RoboDK station: Stringer B-Bot1-BOX1.rdk

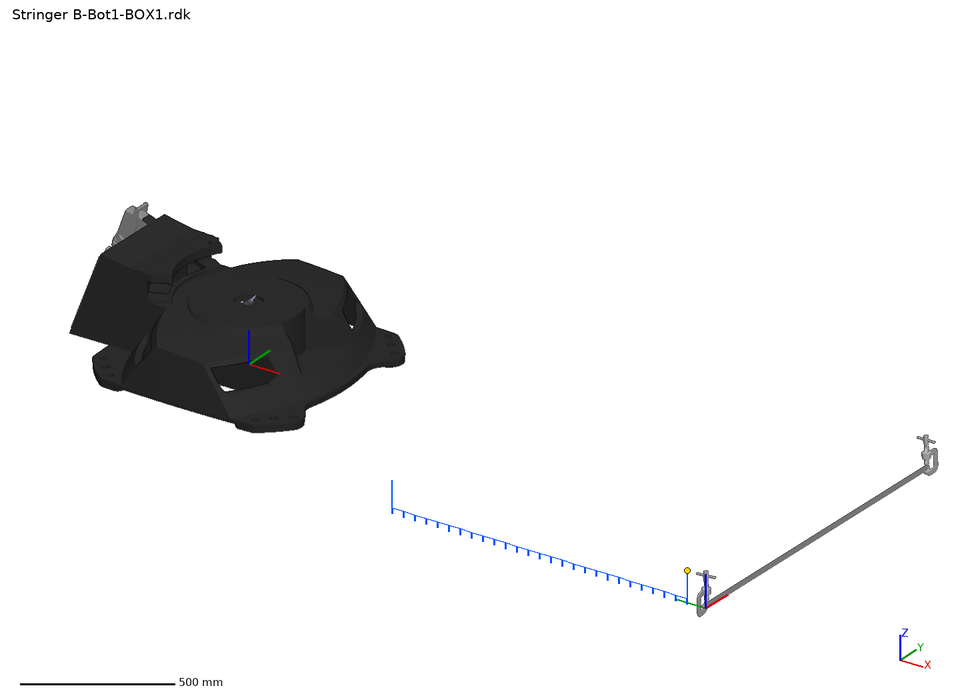
[picture v0: the station drawn from its stored meshes, robots at their saved joint values, targets as dots, program paths as lines]
Station Stringer B-Bot1-BOX1 (saved by RoboDK 5.2.3). Poses are relative to the parent item; angles as X-Y-Z fixed-axis rotations.
  - frame KUKA KR 210 R2700 extra Base at (0, 0, 0) mm
    - robot KUKA KR 210 R2700 extra: 6 axes, payload 210 kg, reach 2696 mm, repeatability 0.06 mm, weight 1068 kg
        joint limits [-185, -140, -120, -350, -125, -350] to [185, -5, 155, 350, 125, 350]; home [0, -90, 90, 0, 0, 0]; saved at [-38.984, -26.717, 86.283, 94.063, 23.385, -126.593]
      - tool Spindle, TCP at (32, 0, 260) mm, rotated rx 0 ry 39 rz 0 deg, size 157.3 x 72 x 259.9 mm
  - frame Frame 2 at (1800, 0, -372.68) mm, rotated rx 0 ry 0 rz 90 deg
    - object STringer B-Bot1-BOX1 at (0, 0, 0) mm, rotated rx 0 ry 0 rz -90 deg, 27 curves, geometry from Point 27
    - object L-Stringer B - Bot1-BOX1 at (0, 0, 0) mm, size 1250 x 20 x 20 mm, geometry from L-Stringer B - Bot1-BOX1.stl
  - machining project Point settings: rotZ(0) | rotX(0)*rotY(0) | rotz(0) | onStart | onPathStart | onApproach | onPoint | onRetract | onFinish | SetRPM(%1) | SetTool(%1) | Extruder(%1) | default | default | OutOnMov(%1) | OutOffMov(%1) | onPathFinish | M_RunCode(%1)
  - program Point (146 instructions, listed below)
  - object FinalClamp at (1791.3, 1250.9, -313.4) mm, rotated rx 0 ry 88.39 rz 0 deg, size 145.3 x 71.1 x 72 mm, geometry from FinalClamp.stp
  - object FinalClamp2 at (1785.63, 21.46, -310.92) mm, rotated rx 159.55 ry 88.7 rz -13.81 deg, size 145.3 x 71.1 x 72 mm, geometry from FinalClamp.stp
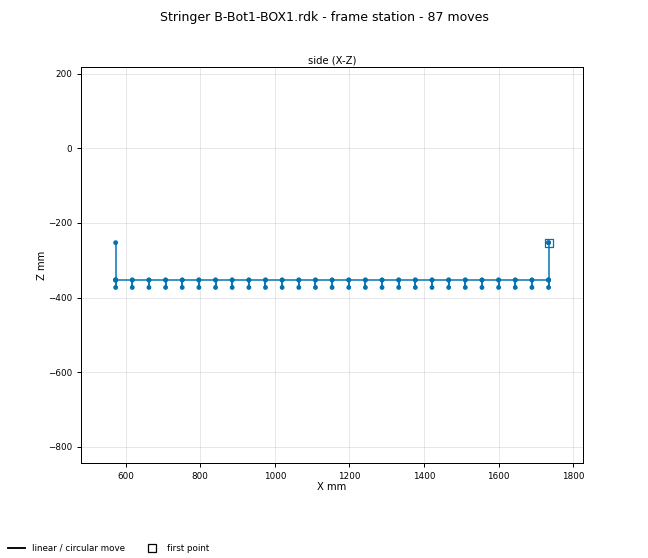
[picture p0: tool path of Stringer B-Bot1-BOX1.rdk in frame station, 87 of 87 moves have a stored position in this frame; points joined in program order, loops and branches not executed]

--- program Point (robot KUKA KR 210 R2700 extra) ---
  Smooth(1)
  Set speed (1000.0 mm/s)
  Set Ref.: Frame 2
  Set Tool: Spindle
  Show Spindle
  MoveJ 1 to (-10.37, 66.57, 120) mm, rotated rx 180 ry 0 rz 180 deg; joints [-2.515, -34.004, 111.796, 176.49, 26.808, -178.821]
  MoveL 2 to (-10.37, 66.57, 120) mm, rotated rx 180 ry 0 rz 180 deg; joints [-2.515, -34.004, 111.796, 176.49, 26.808, -178.821]
  MoveL 3 to (-10.37, 66.57, 20) mm, rotated rx -180 ry 0 rz -180 deg; joints [-2.515, -28.677, 109.154, 176.784, 29.489, -179.155]
  MoveL 4 to (-10.37, 66.57, 20) mm, rotated rx -180 ry 0 rz -180 deg; joints [-2.515, -28.677, 109.154, 176.784, 29.489, -179.155]
  Set speed (50.0 mm/s)
  MoveL 5 to (-10.37, 66.57, 0) mm, rotated rx 180 ry 0 rz 180 deg; joints [-2.515, -27.619, 108.578, 176.831, 29.97, -179.209]
  MoveL 6 to (-10.37, 66.57, 20) mm, rotated rx -180 ry 0 rz -180 deg; joints [-2.515, -28.677, 109.154, 176.784, 29.489, -179.155]
  Set speed (1000.0 mm/s)
  MoveL 7 to (-10.37, 111.19, 20) mm, rotated rx -180 ry 0 rz -180 deg; joints [-4.196, -28.658, 109.018, 174.617, 29.393, -178.57]
  Set speed (50.0 mm/s)
  MoveL 8 to (-10.37, 111.19, 0) mm, rotated rx -180 ry 0 rz -180 deg; joints [-4.196, -27.602, 108.443, 174.695, 29.872, -178.66]
  MoveL 9 to (-10.37, 111.19, 20) mm, rotated rx -180 ry 0 rz -180 deg; joints [-4.196, -28.658, 109.018, 174.617, 29.393, -178.57]
  Set speed (1000.0 mm/s)
  MoveL 10 to (-10.37, 155.8, 20) mm, rotated rx -180 ry 0 rz -180 deg; joints [-5.869, -28.63, 108.815, 172.432, 29.251, -177.955]
  Set speed (50.0 mm/s)
  MoveL 11 to (-10.37, 155.8, 0) mm, rotated rx -180 ry 0 rz -180 deg; joints [-5.869, -27.576, 108.24, 172.543, 29.727, -178.083]
  MoveL 12 to (-10.37, 155.8, 20) mm, rotated rx -180 ry 0 rz -180 deg; joints [-5.869, -28.63, 108.815, 172.432, 29.251, -177.955]
  Set speed (1000.0 mm/s)
  MoveL 13 to (-10.37, 200.42, 20) mm, rotated rx 180 ry 0 rz 180 deg; joints [-7.533, -28.592, 108.543, 170.222, 29.064, -177.301]
  Set speed (50.0 mm/s)
  MoveL 14 to (-10.37, 200.42, 0) mm, rotated rx 180 ry 0 rz 180 deg; joints [-7.533, -27.54, 107.97, 170.365, 29.535, -177.466]
  MoveL 15 to (-10.37, 200.42, 20) mm, rotated rx 180 ry 0 rz 180 deg; joints [-7.533, -28.592, 108.543, 170.222, 29.064, -177.301]
  Set speed (1000.0 mm/s)
  MoveL 16 to (-10.37, 245.03, 20) mm, rotated rx -180 ry 0 rz -180 deg; joints [-9.184, -28.542, 108.204, 167.979, 28.834, -176.595]
  Set speed (50.0 mm/s)
  MoveL 17 to (-10.37, 245.03, 0) mm, rotated rx -180 ry 0 rz -180 deg; joints [-9.184, -27.493, 107.632, 168.157, 29.301, -176.798]
  MoveL 18 to (-10.37, 245.03, 20) mm, rotated rx -180 ry 0 rz -180 deg; joints [-9.184, -28.542, 108.204, 167.979, 28.834, -176.595]
  Set speed (1000.0 mm/s)
  MoveL 19 to (-10.37, 289.65, 20) mm, rotated rx 180 ry 0 rz 180 deg; joints [-10.82, -28.481, 107.797, 165.696, 28.566, -175.826]
  Set speed (50.0 mm/s)
  MoveL 20 to (-10.37, 289.65, 0) mm, rotated rx 180 ry 0 rz -180 deg; joints [-10.82, -27.436, 107.226, 165.908, 29.026, -176.068]
  MoveL 21 to (-10.37, 289.65, 20) mm, rotated rx 180 ry 0 rz 180 deg; joints [-10.82, -28.481, 107.797, 165.696, 28.566, -175.826]
  Set speed (1000.0 mm/s)
  MoveL 22 to (-10.37, 334.26, 20) mm, rotated rx 180 ry 0 rz 180 deg; joints [-12.437, -28.407, 107.323, 163.366, 28.261, -174.983]
  Set speed (50.0 mm/s)
  MoveL 23 to (-10.37, 334.26, 0) mm, rotated rx -180 ry 0 rz -180 deg; joints [-12.437, -27.366, 106.754, 163.613, 28.714, -175.264]
  MoveL 24 to (-10.37, 334.26, 20) mm, rotated rx 180 ry 0 rz 180 deg; joints [-12.437, -28.407, 107.323, 163.366, 28.261, -174.983]
  Set speed (1000.0 mm/s)
  MoveL 25 to (-10.37, 378.88, 20) mm, rotated rx -180 ry 0 rz -180 deg; joints [-14.036, -28.32, 106.782, 160.98, 27.925, -174.054]
  Set speed (50.0 mm/s)
  MoveL 26 to (-10.37, 378.88, 0) mm, rotated rx -180 ry 0 rz -180 deg; joints [-14.036, -27.283, 106.214, 161.263, 28.369, -174.376]
  MoveL 27 to (-10.37, 378.88, 20) mm, rotated rx -180 ry 0 rz -180 deg; joints [-14.036, -28.32, 106.782, 160.98, 27.925, -174.054]
  Set speed (1000.0 mm/s)
  MoveL 28 to (-10.37, 423.5, 20) mm, rotated rx -180 ry 0 rz -180 deg; joints [-15.612, -28.217, 106.174, 158.529, 27.562, -173.029]
  Set speed (50.0 mm/s)
  MoveL 29 to (-10.37, 423.5, 0) mm, rotated rx -180 ry 0 rz -180 deg; joints [-15.612, -27.186, 105.608, 158.851, 27.996, -173.393]
  MoveL 30 to (-10.37, 423.5, 20) mm, rotated rx -180 ry 0 rz -180 deg; joints [-15.612, -28.217, 106.174, 158.529, 27.562, -173.029]
  Set speed (1000.0 mm/s)
  MoveL 31 to (-10.37, 468.11, 20) mm, rotated rx 180 ry 0 rz -180 deg; joints [-17.164, -28.099, 105.499, 156.008, 27.177, -171.897]
  Set speed (50.0 mm/s)
  MoveL 32 to (-10.37, 468.11, 0) mm, rotated rx 180 ry 0 rz 180 deg; joints [-17.164, -27.073, 104.936, 156.368, 27.6, -172.303]
  MoveL 33 to (-10.37, 468.11, 20) mm, rotated rx 180 ry 0 rz -180 deg; joints [-17.164, -28.099, 105.499, 156.008, 27.177, -171.897]
  Set speed (1000.0 mm/s)
  MoveL 34 to (-10.37, 512.73, 20) mm, rotated rx 180 ry 0 rz 180 deg; joints [-18.691, -27.963, 104.758, 153.406, 26.776, -170.648]
  Set speed (50.0 mm/s)
  MoveL 35 to (-10.37, 512.73, 0) mm, rotated rx 180 ry 0 rz 180 deg; joints [-18.691, -26.943, 104.197, 153.806, 27.187, -171.097]
  MoveL 36 to (-10.37, 512.73, 20) mm, rotated rx 180 ry 0 rz 180 deg; joints [-18.691, -27.963, 104.758, 153.406, 26.776, -170.648]
  Set speed (1000.0 mm/s)
  MoveL 37 to (-10.37, 557.34, 20) mm, rotated rx 180 ry 0 rz -180 deg; joints [-20.191, -27.808, 103.95, 150.716, 26.364, -169.271]
  Set speed (50.0 mm/s)
  MoveL 38 to (-10.37, 557.34, 0) mm, rotated rx 180 ry 0 rz 180 deg; joints [-20.191, -26.795, 103.392, 151.158, 26.761, -169.765]
  MoveL 39 to (-10.37, 557.34, 20) mm, rotated rx 180 ry 0 rz -180 deg; joints [-20.191, -27.808, 103.95, 150.716, 26.364, -169.271]
  Set speed (1000.0 mm/s)
  MoveL 40 to (-10.37, 601.96, 20) mm, rotated rx -180 ry 0 rz -180 deg; joints [-21.662, -27.633, 103.077, 147.932, 25.947, -167.758]
  Set speed (50.0 mm/s)
  MoveL 41 to (-10.37, 601.96, 0) mm, rotated rx 180 ry 0 rz -180 deg; joints [-21.662, -26.627, 102.521, 148.415, 26.329, -168.297]
  MoveL 42 to (-10.37, 601.96, 20) mm, rotated rx -180 ry 0 rz -180 deg; joints [-21.662, -27.633, 103.077, 147.932, 25.947, -167.758]
  Set speed (1000.0 mm/s)
  MoveL 43 to (-10.37, 646.57, 20) mm, rotated rx -180 ry 0 rz -180 deg; joints [-23.104, -27.437, 102.138, 145.046, 25.533, -166.101]
  Set speed (50.0 mm/s)
  MoveL 44 to (-10.37, 646.57, 0) mm, rotated rx 180 ry 0 rz 180 deg; joints [-23.104, -26.438, 101.584, 145.572, 25.899, -166.685]
  MoveL 45 to (-10.37, 646.57, 20) mm, rotated rx -180 ry 0 rz -180 deg; joints [-23.104, -27.437, 102.138, 145.046, 25.533, -166.101]
  Set speed (1000.0 mm/s)
  MoveL 46 to (-10.37, 691.19, 20) mm, rotated rx -180 ry 0 rz 180 deg; joints [-24.516, -27.218, 101.133, 142.051, 25.128, -164.292]
  Set speed (50.0 mm/s)
  MoveL 47 to (-10.37, 691.19, 0) mm, rotated rx 180 ry 0 rz 180 deg; joints [-24.516, -26.226, 100.581, 142.62, 25.476, -164.921]
  MoveL 48 to (-10.37, 691.19, 20) mm, rotated rx -180 ry 0 rz 180 deg; joints [-24.516, -27.218, 101.133, 142.051, 25.128, -164.292]
  Set speed (1000.0 mm/s)
  MoveL 49 to (-10.37, 735.8, 20) mm, rotated rx 180 ry 0 rz 180 deg; joints [-25.896, -26.974, 100.063, 138.945, 24.739, -162.327]
  Set speed (50.0 mm/s)
  MoveL 50 to (-10.37, 735.8, 0) mm, rotated rx 180 ry 0 rz -180 deg; joints [-25.896, -25.99, 99.513, 139.557, 25.068, -163]
  MoveL 51 to (-10.37, 735.8, 20) mm, rotated rx 180 ry 0 rz 180 deg; joints [-25.896, -26.974, 100.063, 138.945, 24.739, -162.327]
  Set speed (1000.0 mm/s)
  MoveL 52 to (-10.37, 780.42, 20) mm, rotated rx -180 ry 0 rz -180 deg; joints [-27.245, -26.705, 98.926, 135.724, 24.374, -160.201]
  Set speed (50.0 mm/s)
  MoveL 53 to (-10.37, 780.42, 0) mm, rotated rx 180 ry 0 rz -180 deg; joints [-27.245, -25.729, 98.379, 136.376, 24.683, -160.918]
  MoveL 54 to (-10.37, 780.42, 20) mm, rotated rx -180 ry 0 rz -180 deg; joints [-27.245, -26.705, 98.926, 135.724, 24.374, -160.201]
  Set speed (1000.0 mm/s)
  MoveL 55 to (-10.37, 825.03, 20) mm, rotated rx 180 ry 0 rz -180 deg; joints [-28.562, -26.409, 97.724, 132.388, 24.04, -157.915]
  Set speed (50.0 mm/s)
  MoveL 56 to (-10.37, 825.03, 0) mm, rotated rx 180 ry 0 rz 180 deg; joints [-28.562, -25.441, 97.179, 133.08, 24.327, -158.673]
  MoveL 57 to (-10.37, 825.03, 20) mm, rotated rx 180 ry 0 rz -180 deg; joints [-28.562, -26.409, 97.724, 132.388, 24.04, -157.915]
  Set speed (1000.0 mm/s)
  MoveL 58 to (-10.37, 869.65, 20) mm, rotated rx 180 ry 0 rz 180 deg; joints [-29.848, -26.084, 96.456, 128.938, 23.745, -155.469]
  Set speed (50.0 mm/s)
  MoveL 59 to (-10.37, 869.65, 0) mm, rotated rx 180 ry 0 rz 180 deg; joints [-29.848, -25.124, 95.912, 129.666, 24.009, -156.265]
  MoveL 60 to (-10.37, 869.65, 20) mm, rotated rx 180 ry 0 rz 180 deg; joints [-29.848, -26.084, 96.456, 128.938, 23.745, -155.469]
  Set speed (1000.0 mm/s)
  MoveL 61 to (-10.37, 914.26, 20) mm, rotated rx 180 ry 0 rz 180 deg; joints [-31.1, -25.73, 95.121, 125.38, 23.497, -152.87]
  Set speed (50.0 mm/s)
  MoveL 62 to (-10.37, 914.26, 0) mm, rotated rx 180 ry 0 rz -180 deg; joints [-31.1, -24.778, 94.579, 126.141, 23.736, -153.7]
  MoveL 63 to (-10.37, 914.26, 20) mm, rotated rx 180 ry 0 rz 180 deg; joints [-31.1, -25.73, 95.121, 125.38, 23.497, -152.87]
  Set speed (1000.0 mm/s)
  MoveL 64 to (-10.37, 958.88, 20) mm, rotated rx 180 ry 0 rz -180 deg; joints [-32.321, -25.344, 93.719, 121.722, 23.301, -150.125]
  Set speed (50.0 mm/s)
  MoveL 65 to (-10.37, 958.88, 0) mm, rotated rx 180 ry 0 rz 180 deg; joints [-32.321, -24.4, 93.179, 122.511, 23.516, -150.985]
  MoveL 66 to (-10.37, 958.88, 20) mm, rotated rx 180 ry 0 rz -180 deg; joints [-32.321, -25.344, 93.719, 121.722, 23.301, -150.125]
  Set speed (1000.0 mm/s)
  MoveL 67 to (-10.37, 1003.5, 20) mm, rotated rx 180 ry 0 rz 180 deg; joints [-33.51, -24.925, 92.249, 117.977, 23.167, -147.248]
  Set speed (50.0 mm/s)
  MoveL 68 to (-10.37, 1003.5, 0) mm, rotated rx 180 ry 0 rz 180 deg; joints [-33.51, -23.99, 91.71, 118.788, 23.355, -148.13]
  MoveL 69 to (-10.37, 1003.5, 20) mm, rotated rx 180 ry 0 rz 180 deg; joints [-33.51, -24.925, 92.249, 117.977, 23.167, -147.248]
  Set speed (1000.0 mm/s)
  MoveL 70 to (-10.37, 1048.11, 20) mm, rotated rx 180 ry 0 rz 180 deg; joints [-34.666, -24.472, 90.71, 114.162, 23.099, -144.255]
  Set speed (50.0 mm/s)
  MoveL 71 to (-10.37, 1048.11, 0) mm, rotated rx -180 ry 0 rz -180 deg; joints [-34.666, -23.545, 90.172, 114.987, 23.261, -145.153]
  MoveL 72 to (-10.37, 1048.11, 20) mm, rotated rx 180 ry 0 rz 180 deg; joints [-34.666, -24.472, 90.71, 114.162, 23.099, -144.255]
  Set speed (1000.0 mm/s)
  MoveL 73 to (-10.37, 1092.73, 20) mm, rotated rx -180 ry 0 rz -180 deg; joints [-35.792, -23.984, 89.102, 110.293, 23.104, -141.164]
  Set speed (50.0 mm/s)
  MoveL 74 to (-10.37, 1092.73, 0) mm, rotated rx -180 ry 0 rz -180 deg; joints [-35.792, -23.065, 88.563, 111.125, 23.239, -142.069]
  MoveL 75 to (-10.37, 1092.73, 20) mm, rotated rx -180 ry 0 rz -180 deg; joints [-35.792, -23.984, 89.102, 110.293, 23.104, -141.164]
  Set speed (1000.0 mm/s)
  MoveL 76 to (-10.37, 1137.34, 20) mm, rotated rx 180 ry 0 rz -180 deg; joints [-36.886, -23.459, 87.421, 106.394, 23.187, -137.998]
  Set speed (50.0 mm/s)
  MoveL 77 to (-10.37, 1137.34, 0) mm, rotated rx 180 ry 0 rz 180 deg; joints [-36.886, -22.548, 86.883, 107.225, 23.295, -138.903]
  MoveL 78 to (-10.37, 1137.34, 20) mm, rotated rx 180 ry 0 rz -180 deg; joints [-36.886, -23.459, 87.421, 106.394, 23.187, -137.998]
  Set speed (1000.0 mm/s)
  MoveL 79 to (-10.37, 1181.96, 20) mm, rotated rx 180 ry 0 rz -180 deg; joints [-37.95, -22.895, 85.667, 102.486, 23.353, -134.78]
  Set speed (50.0 mm/s)
  MoveL 80 to (-10.37, 1181.96, 0) mm, rotated rx -180 ry 0 rz -180 deg; joints [-37.95, -21.991, 85.129, 103.308, 23.434, -135.676]
  MoveL 81 to (-10.37, 1181.96, 20) mm, rotated rx 180 ry 0 rz -180 deg; joints [-37.95, -22.895, 85.667, 102.486, 23.353, -134.78]
  Set speed (1000.0 mm/s)
  MoveL 82 to (-10.37, 1226.57, 20) mm, rotated rx 180 ry 0 rz 180 deg; joints [-38.984, -22.29, 83.838, 98.596, 23.603, -131.536]
  Set speed (50.0 mm/s)
  MoveL 83 to (-10.37, 1226.57, 0) mm, rotated rx -180 ry 0 rz -180 deg; joints [-38.984, -21.394, 83.298, 99.4, 23.659, -132.414]
  MoveL 84 to (-10.37, 1226.57, 20) mm, rotated rx 180 ry 0 rz 180 deg; joints [-38.984, -22.29, 83.838, 98.596, 23.603, -131.536]
  MoveL 85 to (-10.37, 1226.57, 20) mm, rotated rx 180 ry 0 rz 180 deg; joints [-38.984, -22.29, 83.838, 98.596, 23.603, -131.536]
  Set speed (1000.0 mm/s)
  MoveL 86 to (-10.37, 1226.57, 20) mm, rotated rx 180 ry 0 rz 180 deg; joints [-38.984, -22.29, 83.838, 98.596, 23.603, -131.536]
  MoveL 87 to (-10.37, 1226.57, 120) mm, rotated rx 180 ry 0 rz 180 deg; joints [-38.984, -26.717, 86.283, 94.063, 23.385, -126.593]
